{attribute 'qualified_only'}
VAR_GLOBAL
	eenHzTrigger : BOOL;
END_VAR

(* stored: Version 1.1.0.1, ProductVersion 3.1.4024.12
   GVL DB2_Counters: Id {a7503705-2eae-4ce4-bf29-6bfcd897118d} *)
